Fanuc KAREL source: FORCE_SPMENU.kl

PROGRAM T
%NOLOCKGROUP
VAR
 v0 : INTEGER
 v1 : INTEGER
 v2 : INTEGER
BEGIN
 FORCE_SPMENU(v0, v1, v2)
END T
